FUNCTION_BLOCK AX_AE_MERGE (* Merges an AE (Event only) and an AX (Event + BOOL) adapter. Output is AX with BOOL from IN_AX. *)
  (* Standard: 61499-2; Description: Copyright (c) 2026 HR Agrartechnik GmbH This program and the accompanying materials are made available under the terms of the Eclipse Public License 2.0 which is available at https://www.eclipse.org/legal/epl-2.0/ SPDX-License-Identifier: EPL-2.0 *)
  (* Version 1.0, 2026-01-17, Franz Höpfinger, HR Agrartechnik GmbH *)
  PACKAGE adapter::events::unidirectional;
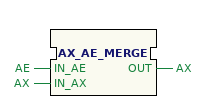
  SOCKETS
    IN_AE : adapter::types::unidirectional::AE; (* AE Signal (Events only) *)
    IN_AX : adapter::types::unidirectional::AX; (* Main AX Signal (Events + Data) *)
  END_SOCKETS
  PLUGS
    OUT : adapter::types::unidirectional::AX; (* Merged AX Output *)
  END_PLUGS
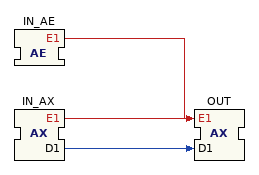
  EVENT_CONNECTIONS
    IN_AX.E1 TO OUT.E1;
    IN_AE.E1 TO OUT.E1;
  END_CONNECTIONS
  DATA_CONNECTIONS
    IN_AX.D1 TO OUT.D1;
  END_CONNECTIONS
END_FUNCTION_BLOCK
